
FUNCTION CB_bool_to_dint : DINT


TITLE = ' Convert a boolean into an double integer '
VERSION : '1.0'
AUTHOR  : CB
NAME    : boToDint
FAMILY  : TNI

VAR_INPUT
    IN : BOOL;
END_VAR

VAR_TEMP

END_VAR

BEGIN

CB_bool_to_dint := BOOL_TO_DINT(IN);

END_FUNCTION
